// TIA Portal V15.1 export
// export: Created 2024-06-21T08:40:52.5067836Z, ExportSetting WithDefaults, DisplayName Totally Integrated Automation Portal, DisplayVersion V15.1 Update 5, DisplayName TIA Portal Openness, DisplayVersion V15.1 Update 5, DisplayName SINAMICS Startdrive Advanced, DisplayVersion V15.1, DisplayName G130, G150, S120, S150, SINAMICS MV, S210, DisplayVersion V15.1, DisplayName G110M, G120, G120C, G120D, G120P, DisplayVersion V15.1, DisplayName STEP 7 Professional, DisplayVersion V15.1 Update 5, DisplayName STEP 7 Safety, DisplayVersion V15.1, DisplayName WinCC Professional, DisplayVersion V15.1 Update 5, DisplayName SIMATIC Visualization Architect, DisplayVersion V15.1
FUNCTION_BLOCK "LAcofDet"   // FB1416, FBD
TITLE = LAcofDet
{ S7_Optimized_Access := 'FALSE' }
AUTHOR : VCC
FAMILY : Actuator
NAME : LAcofDet
VERSION : 1.0
// ===============================================================================
// This module handles a partdetection with all his functions and alarms
// Functions are DetCheckOn, DetCheckOff and EnableAlarm
// Outputs are DetAlarm and DetSim signal
// ===============================================================================
// stored: AutoNumber false, IsIECCheckEnabled false, SetENOAutomatically False, UDAEnableTagReadback false
   VAR_INPUT
      I_Input { ExternalAccessible := 'False'; ExternalVisible := 'False'; ExternalWritable := 'False'} : Bool;   // Actual input from sensor
      I_SignalCheckOn { ExternalAccessible := 'False'; ExternalVisible := 'False'; ExternalWritable := 'False'} : Bool;   // Signal to check signal is on
      I_SignalCheckOff { ExternalAccessible := 'False'; ExternalVisible := 'False'; ExternalWritable := 'False'} : Bool;   // Signal to check signal is off
      I_MaxAcofTime { ExternalAccessible := 'False'; ExternalVisible := 'False'; ExternalWritable := 'False'} : DInt;   // Maximum Time (ms) that the function may run (create overtime)
      I_AlarmClass { ExternalAccessible := 'False'; ExternalVisible := 'False'; ExternalWritable := 'False'} : Char;   // Alarm class -> A - B - C - D or E
      I_EnableAlarm { ExternalAccessible := 'False'; ExternalVisible := 'False'; ExternalWritable := 'False'} : Bool;   // Enable alarms
      I_Simulate { ExternalAccessible := 'False'; ExternalVisible := 'False'; ExternalWritable := 'False'} : Bool;   // Simulate modus
      I_AlarmResetPB { ExternalAccessible := 'False'; ExternalVisible := 'False'; ExternalWritable := 'False'} : Bool;   // Alarm reset pushbutton is activated
      I_Invisible { ExternalAccessible := 'False'; ExternalVisible := 'False'; ExternalWritable := 'False'} : Bool;   // Invisible
      C_DisableViaHMI { ExternalAccessible := 'False'; ExternalVisible := 'False'; ExternalWritable := 'False'} : Bool;   // Config to enable/disable the detection via the HMI
   END_VAR
   VAR_OUTPUT
      O_DetOn { ExternalAccessible := 'False'; ExternalVisible := 'False'; ExternalWritable := 'False'} : Bool;   // Detection signal to use in program
      O_Alarm { ExternalAccessible := 'False'; ExternalVisible := 'False'; ExternalWritable := 'False'} : Bool;   // Detection alarm
      O_AlarmABCondition { ExternalAccessible := 'False'; ExternalVisible := 'False'; ExternalWritable := 'False'} : Bool;   // Alarm AB condition
      O_AlarmDisabled { ExternalAccessible := 'False'; ExternalVisible := 'False'; ExternalWritable := 'False'} : Bool;   // Alarm disabled from HMI
      H_IAnim { ExternalAccessible := 'False'; ExternalVisible := 'False'; ExternalWritable := 'False'} : DWord;   // For animation of the icon
   END_VAR
   VAR DB_SPECIFIC
      H_In : Struct   // HMI
         DisableAlarm : Bool;   // Disable alarm from HMI
      END_STRUCT;
      H_Out : Struct   // HMI
         Anim : Word;   // HMI Animation of the object
         DBnr : Int;   // HMI Animation DB number
      END_STRUCT;
      DetOn { ExternalAccessible := 'False'; ExternalVisible := 'False'; ExternalWritable := 'False'} : Bool;   // Static variable of O_DetOn
      DetOvtAlarm { ExternalAccessible := 'False'; ExternalVisible := 'False'; ExternalWritable := 'False'} : Bool;   // Static variable of O_DetAlarm
      Alarm { ExternalAccessible := 'False'; ExternalVisible := 'False'; ExternalWritable := 'False'} : Bool;   // Alarm condition
      AlarmDisabled { ExternalAccessible := 'False'; ExternalVisible := 'False'; ExternalWritable := 'False'} : Bool;   // Alarm disabled from HMI
      AlarmClass_A { ExternalAccessible := 'False'; ExternalVisible := 'False'; ExternalWritable := 'False'} : Bool;   // The alarm is from alarm class A
      AlarmClass_B { ExternalAccessible := 'False'; ExternalVisible := 'False'; ExternalWritable := 'False'} : Bool;   // The alarm is from alarm class B
      AlarmClass_C { ExternalAccessible := 'False'; ExternalVisible := 'False'; ExternalWritable := 'False'} : Bool;   // The alarm is from alarm class C
      AlarmClass_D { ExternalAccessible := 'False'; ExternalVisible := 'False'; ExternalWritable := 'False'} : Bool;   // The alarm is from alarm class D
      AlarmClass_E { ExternalAccessible := 'False'; ExternalVisible := 'False'; ExternalWritable := 'False'} : Bool;   // The alarm is from alarm class E
      DBnr { ExternalAccessible := 'False'; ExternalVisible := 'False'; ExternalWritable := 'False'} : Int;   // HMI DB number
   END_VAR
   VAR
      MaxTimeTimer { ExternalAccessible := 'False'; ExternalVisible := 'False'; ExternalWritable := 'False'; S7_SetPoint := 'True'} : "LTimer";   // Creating alarm overtime
   END_VAR
BEGIN

NETWORK
TITLE = **** 1 - Inputs **** DB number
// DB number
      L     DINO;
      T     #DBnr;

NETWORK
TITLE = **** 1 - Inputs **** Alarm class
// Alarm class
// Alarm class = E
      L     #I_AlarmClass;
      L     'E';
      ==I;
      =     #AlarmClass_E;

// Alarm class = D
      L     #I_AlarmClass;
      L     'D';
      ==I;
      =     #AlarmClass_D;

// Alarm class = C
      L     #I_AlarmClass;
      L     'C';
      ==I;
      =     #AlarmClass_C;

// Alarm class = B
      L     #I_AlarmClass;
      L     'B';
      ==I;
      =     #AlarmClass_B;

// Alarm class = A
      AN    #AlarmClass_B;
      AN    #AlarmClass_C;
      AN    #AlarmClass_D;
      AN    #AlarmClass_E;
      =     #AlarmClass_A;


REGION Network 3: **** 2.2 - Alarms - Alarm generation **** Creating alarm overtime
   // Creating alarm overtime
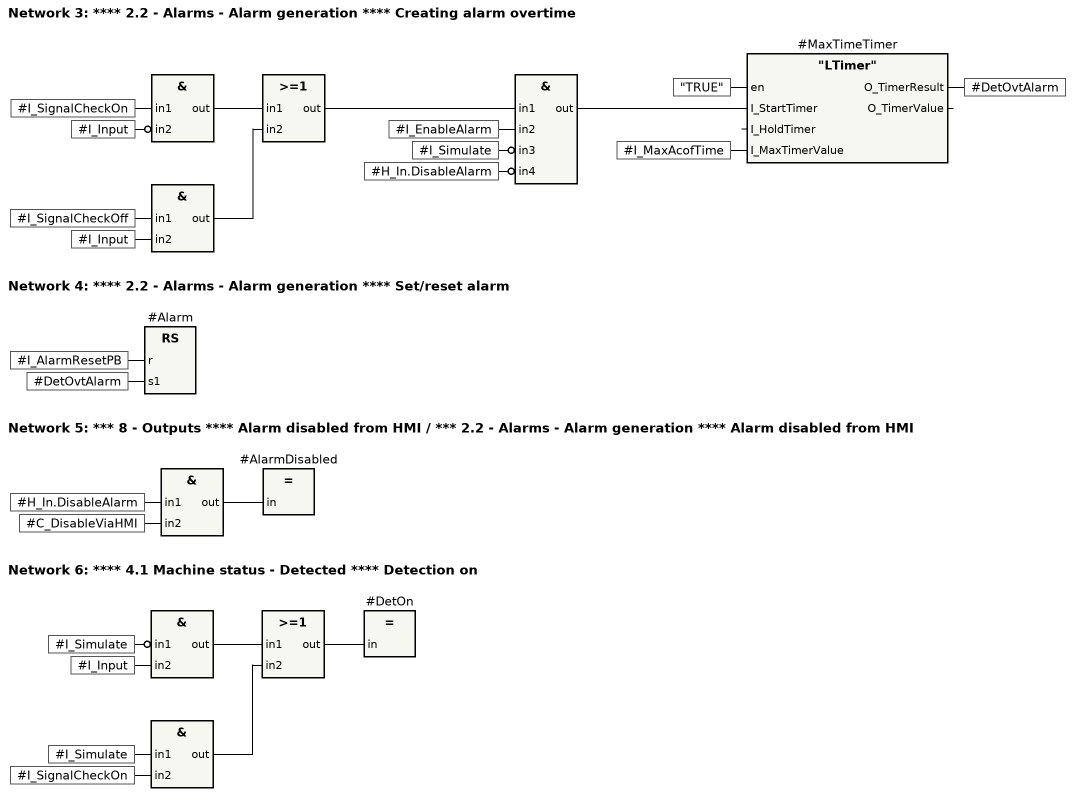
   IF "TRUE" THEN
       #MaxTimeTimer(I_StartTimer := ((#I_SignalCheckOn AND NOT #I_Input) OR (#I_SignalCheckOff AND #I_Input)) AND #I_EnableAlarm AND NOT #I_Simulate AND NOT #H_In.DisableAlarm,   // "LTimer"
                     I_MaxTimerValue := #I_MaxAcofTime,
                     O_TimerResult => #DetOvtAlarm);
   END_IF;
END_REGION

REGION Network 4: **** 2.2 - Alarms - Alarm generation **** Set/reset alarm
   // Set/reset alarm
   IF #I_AlarmResetPB THEN
       #Alarm := FALSE;   // RS flip-flop
   END_IF;
   IF #DetOvtAlarm THEN #Alarm := TRUE; END_IF;
END_REGION

REGION Network 5: *** 8 - Outputs **** Alarm disabled from HMI / *** 2.2 - Alarms - Alarm generation **** Alarm disabled from HMI
   // Alarm disabled from HMI
   #AlarmDisabled := #H_In.DisableAlarm AND #C_DisableViaHMI;
END_REGION

REGION Network 6: **** 4.1 Machine status - Detected **** Detection on
   // Detection on
   #DetOn := (NOT #I_Simulate AND #I_Input) OR (#I_Simulate AND #I_SignalCheckOn);
END_REGION

REGION Network 7: **** 4.6 - Mashine Status - Indications **** Icon Animation
   // Icon Animation
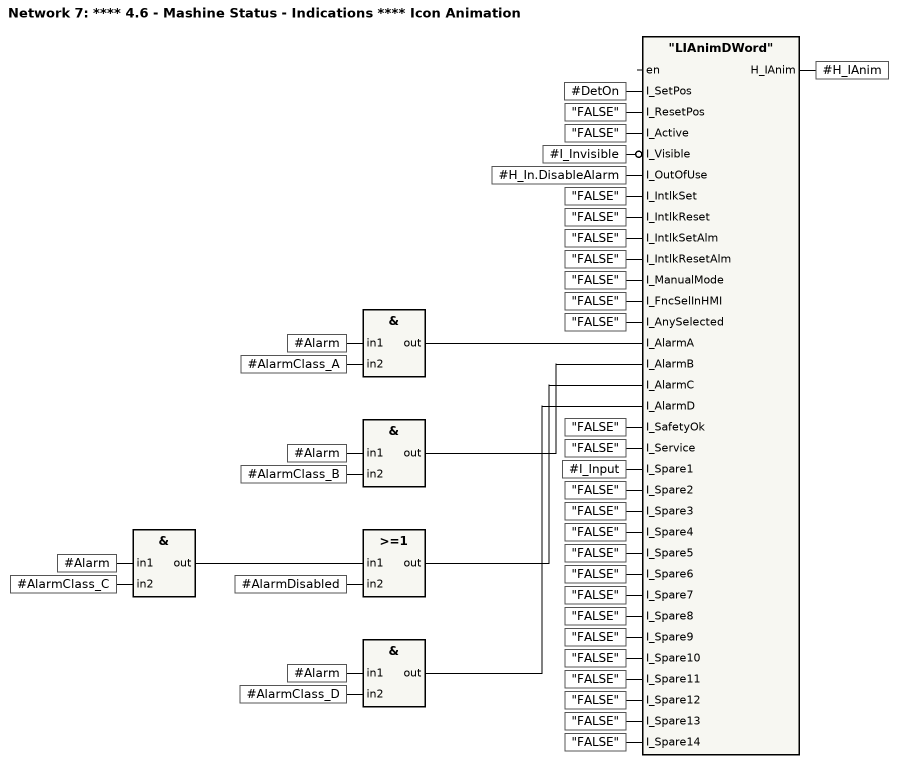
   "LIAnimDWord"(I_SetPos := #DetOn,
                 I_ResetPos := "FALSE",
                 I_Active := "FALSE",
                 I_Visible := NOT #I_Invisible,
                 I_OutOfUse := #H_In.DisableAlarm,
                 I_IntlkSet := "FALSE",
                 I_IntlkReset := "FALSE",
                 I_IntlkSetAlm := "FALSE",
                 I_IntlkResetAlm := "FALSE",
                 I_ManualMode := "FALSE",
                 I_FncSelInHMI := "FALSE",
                 I_AnySelected := "FALSE",
                 I_AlarmA := #Alarm AND #AlarmClass_A,
                 I_AlarmB := #Alarm AND #AlarmClass_B,
                 I_AlarmC := (#Alarm AND #AlarmClass_C) OR #AlarmDisabled,
                 I_AlarmD := #Alarm AND #AlarmClass_D,
                 I_SafetyOk := "FALSE",
                 I_Service := "FALSE",
                 I_Spare1 := #I_Input,
                 I_Spare2 := "FALSE",
                 I_Spare3 := "FALSE",
                 I_Spare4 := "FALSE",
                 I_Spare5 := "FALSE",
                 I_Spare6 := "FALSE",
                 I_Spare7 := "FALSE",
                 I_Spare8 := "FALSE",
                 I_Spare9 := "FALSE",
                 I_Spare10 := "FALSE",
                 I_Spare11 := "FALSE",
                 I_Spare12 := "FALSE",
                 I_Spare13 := "FALSE",
                 I_Spare14 := "FALSE",
                 H_IAnim => #H_IAnim);
END_REGION

REGION Network 8: **** 4.6 - Machine Status - Indications **** Animation
   // Animation
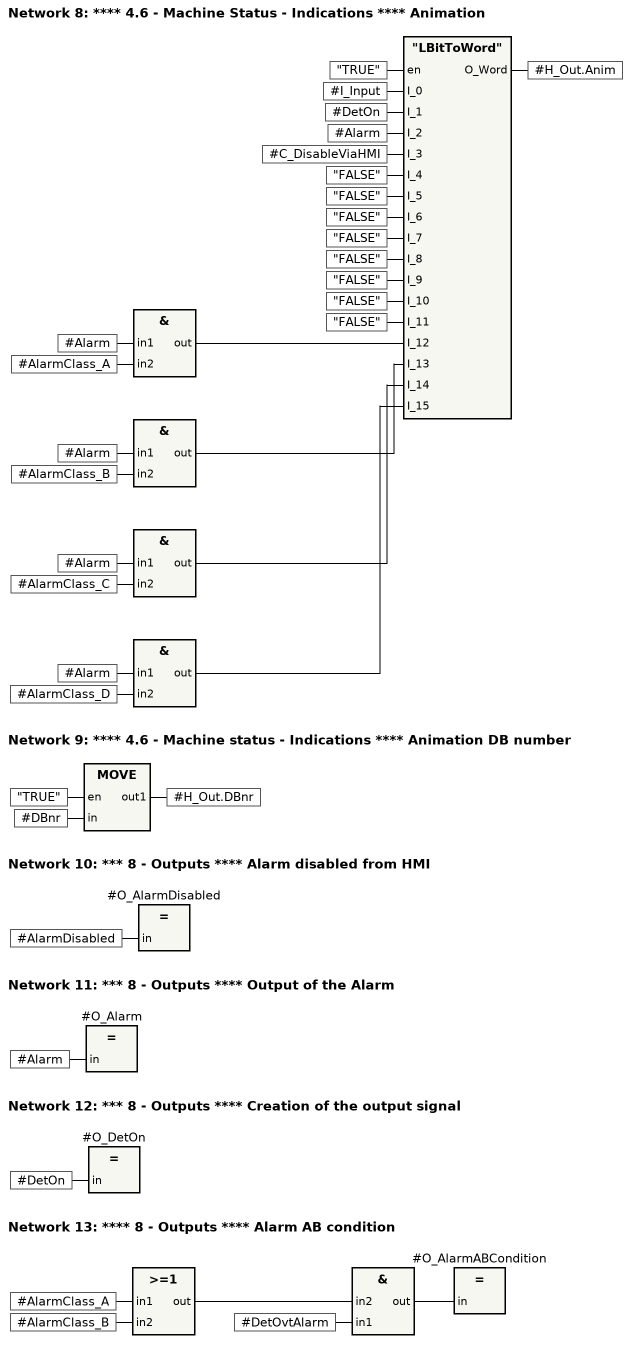
   IF "TRUE" THEN
       "LBitToWord"(I_0 := #I_Input,
                    I_1 := #DetOn,
                    I_2 := #Alarm,
                    I_3 := #C_DisableViaHMI,
                    I_4 := "FALSE",
                    I_5 := "FALSE",
                    I_6 := "FALSE",
                    I_7 := "FALSE",
                    I_8 := "FALSE",
                    I_9 := "FALSE",
                    I_10 := "FALSE",
                    I_11 := "FALSE",
                    I_12 := #Alarm AND #AlarmClass_A,
                    I_13 := #Alarm AND #AlarmClass_B,
                    I_14 := #Alarm AND #AlarmClass_C,
                    I_15 := #Alarm AND #AlarmClass_D,
                    O_Word => #H_Out.Anim);
   END_IF;
END_REGION

REGION Network 9: **** 4.6 - Machine status - Indications **** Animation DB number
   // Animation DB number
   IF "TRUE" THEN #H_Out.DBnr := #DBnr; END_IF;
END_REGION

REGION Network 10: *** 8 - Outputs **** Alarm disabled from HMI
   // Alarm disabled from HMI
   #O_AlarmDisabled := #AlarmDisabled;
END_REGION

REGION Network 11: *** 8 - Outputs **** Output of the Alarm
   // Output of the Alarm
   #O_Alarm := #Alarm;
END_REGION

REGION Network 12: *** 8 - Outputs **** Creation of the output signal
   // Creation of the output signal
   #O_DetOn := #DetOn;
END_REGION

REGION Network 13: **** 8 - Outputs **** Alarm AB condition
   // Alarm AB condition
   #O_AlarmABCondition := (#AlarmClass_A OR #AlarmClass_B) AND #DetOvtAlarm;
END_REGION
END_FUNCTION_BLOCK
